// TIA Portal V17 export
// export: Created 2022-08-15T11:59:21.7814975Z, ExportSetting WithDefaults, DisplayName Totally Integrated Automation Portal, DisplayVersion V17, DisplayName TIA Portal Openness, DisplayVersion V17, DisplayName TIA Portal Version Control Interface, DisplayVersion V17, DisplayName SINAMICS Startdrive Advanced, DisplayVersion V17 Update1, DisplayName SINAMICS Startdrive G110M, G120, G120C, G120D, G120P, G115D, DisplayVersion V17 Update1, DisplayName SINAMICS Startdrive G130, G150, S120, S150, SINAMICS MV, S210, DisplayVersion V17 Update1, DisplayName STEP 7 Professional, DisplayVersion V17, DisplayName STEP 7 Safety, DisplayVersion V17, DisplayName WinCC Advanced, DisplayVersion V17
VAR_GLOBAL   // PLC tag table "Default tag table"
   Sw1 AT %I0.0 : Bool;
   Sw2 AT %I0.1 : Bool;
   Output1 AT %Q0.0 : Bool;
   Output2 AT %Q0.1 : Bool;
   Sw3 AT %I0.2 : Bool;
   Sw4 AT %I0.3 : Bool;
   Sw5 AT %I0.4 : Bool;
   Sw6 AT %I0.5 : Bool;
   Sw7 AT %I0.6 : Bool;
   Sw8 AT %I0.7 : Bool;
   Sw9 AT %I1.0 : Bool;
   Sw10 AT %I1.1 : Bool;
   Output3 AT %Q0.2 : Bool;
   Output4 AT %Q0.3 : Bool;
   Output6 AT %Q0.5 : Bool;
   Sw11 AT %I1.2 : Bool;
   Sw12 AT %I1.3 : Bool;
   Output12 AT %Q0.7 : Bool;
   Output11 AT %Q0.6 : Bool;
   Sw13 AT %I1.4 : Bool;
   Sw14 AT %I1.5 : Bool;
   Output13 AT %Q1.0 : Bool;
   Output14 AT %Q1.1 : Bool;
END_VAR
